VISUALIZATION V_Option6  // 1160x668
END_VISUALIZATION

(* stored: Version 1.1.0.1, ProductVersion 3.1.4024.3
   Visu V_Option6: Id {c26513d2-844e-47f6-8e6a-65159dfdbb6c} *)
